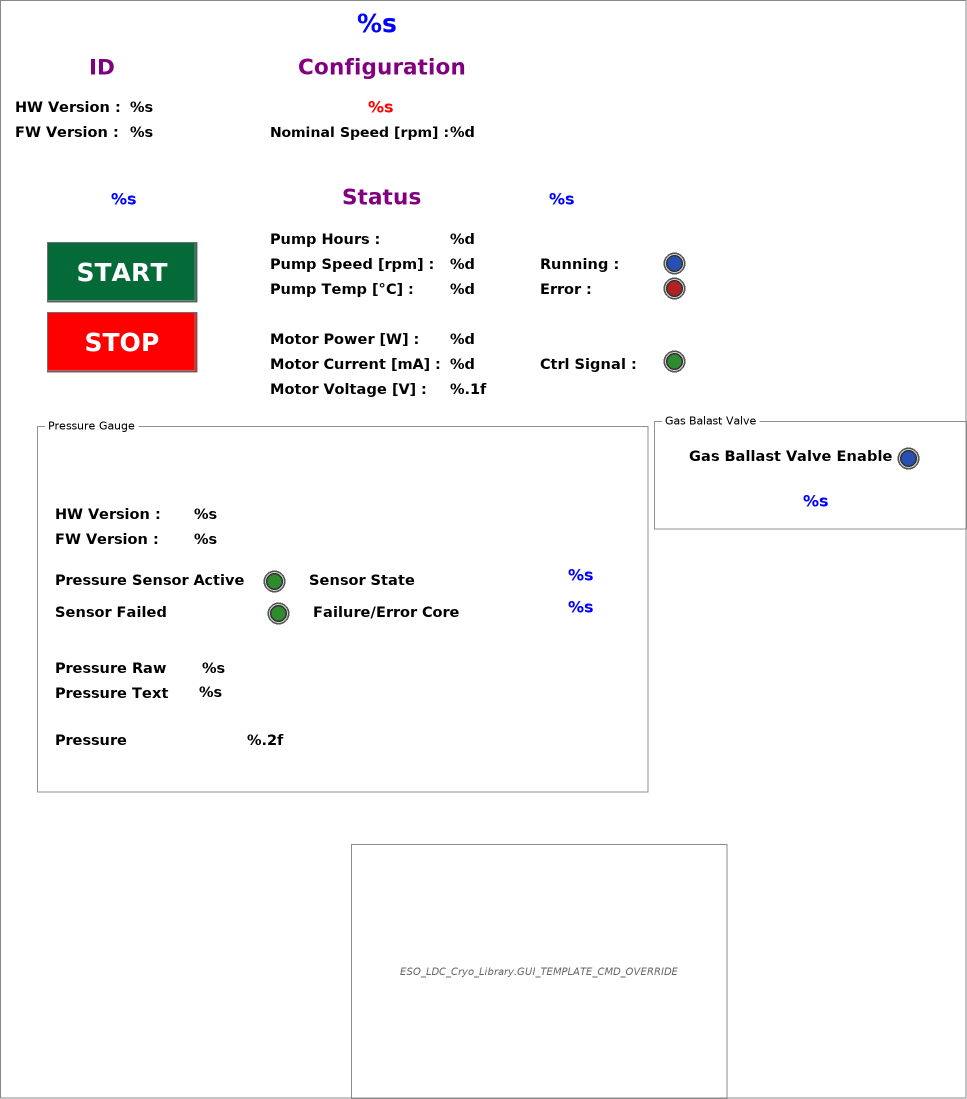
VISUALIZATION TEMPLATE_NOTT_PUMPS  // 967x1099
VAR_IN_OUT
	m_Instance:	FB_NOTT_PUMP_HICUBE_80_NEO;
	m_bEnable:	BOOL;	// Flag to start/stop the pump
	
END_VAR
    Rectangle (27,52 150x30), "ID"
    Rectangle (292,52 180x30), "Configuration"
    Rectangle (307,182 150x30), "Status"
    Lamp1 (662,251 25x25), tooltip "pump speed > 0 rpm", variable: m_Instance.stat.bMoving, style: Lamp-Lamp1-Blue
    Lamp1 (662,276 25x25), tooltip "presence of a warning", variable: m_Instance.stat.bFailure, style: Lamp-Lamp1-Red
    Rectangle (537,249 110x30), "Running :"
    Rectangle (537,274 110x30), "Error :"
    Rectangle (267,117 180x30), "Nominal Speed [rpm] :"
    Rectangle (267,224 180x30), "Pump Hours :"
    Rectangle (447,117 70x30), "%d", text variable: m_Instance.stat.nNominalSpeed
    Rectangle (447,224 70x30), "%d", text variable: m_Instance.stat.nPumpHours
    Rectangle (267,249 180x30), "Pump Speed [rpm] :"
    Rectangle (447,249 70x30), "%d", text variable: m_Instance.stat.nPumpSpeed
    Rectangle (267,274 180x30), "Pump Temp [°C] :"
    Rectangle (447,274 70x30), "%d", text variable: m_Instance.stat.nPumpTemp
    Rectangle (267,349 180x30), "Motor Current [mA] :"
    Rectangle (447,349 70x30), "%d", text variable: m_Instance.stat.nMotorCurr
    Rectangle (267,374 180x30), "Motor Voltage [V] :"
    Rectangle (447,374 70x30), "%.1f", text variable: m_Instance.stat.lrMotorVolt
    Rectangle (262,8 230x30), "%s", text variable: m_Instance.in_sName
    Rectangle (271,92 220x30), "%s", tooltip "Control Mode", text variable: m_Instance.stat.sCtrlViaInt
    Rectangle (127,92 130x30), "%s", tooltip "HW Version", text variable: m_Instance.stat.sHwVersion
    Rectangle (127,117 130x30), "%s", tooltip "FW Version", text variable: m_Instance.stat.sFwVersion
    Button (47,242 150x60), "START"
        OnMouseClick: execute { m_bEnable := TRUE; }
    Button (47,312 150x60), "STOP"
        OnMouseClick: execute { m_bEnable := FALSE; }
    Lamp1 (662,349 25x25), tooltip "If ON, control output signal is active.", variable: m_Instance.q_bStart, style: Lamp-Lamp1-Green
    Rectangle (537,349 110x30), "Ctrl Signal :"
    Rectangle (439,184 246x30), "%s", tooltip "Pump State", text variable: m_Instance.stat.sPumpState
    Rectangle (74,184 100x30), "%s", tooltip "Error Status", text variable: m_Instance.stat.sFailureCode
    Rectangle (267,324 180x30), "Motor Power [W] :"
    Rectangle (447,324 70x30), "%d", text variable: m_Instance.stat.nElecPower
    Rectangle (12,92 110x30), "HW Version :"
    Rectangle (12,117 110x30), "FW Version :"
    Frame (351,844 376x255)
        shows ESO_LDC_Cryo_Library.GUI_TEMPLATE_CMD_OVERRIDE(m_Cmd := MAIN.nott_cryo_ctrl.evac.ctrl.cor_PVP)
    GroupBox (37,418 611x374), "Pressure Gauge"
        Lamp1 (225,151 25x25), tooltip "Pressure Sensor ON", variable: m_Instance.stat.PresSens_bSensorOn, style: Lamp-Lamp1-Green
        Rectangle (15,147 254x30), "Pressure Sensor Active"
        Lamp1 (229,183 25x25), tooltip "Pressure Sensor ON", variable: m_Instance.stat.PresSens_bFailure, style: Lamp-Lamp1-Green
        Rectangle (269,147 254x30), "Sensor State"
        Rectangle (450,174 188x30), "%s", tooltip "Error Status", text variable: m_Instance.stat.PresSens_sFailureCode
        Rectangle (273,179 254x30), "Failure/Error Core"
        Rectangle (15,179 254x30), "Sensor Failed"
        Rectangle (450,142 188x30), "%s", tooltip "Error Status", text variable: m_Instance.stat.PresSens_sSensorState
        Rectangle (15,81 110x30), "HW Version :"
        Rectangle (154,81 130x30), "%s", tooltip "HW Version", text variable: m_Instance.stat.PresSens_sHwVersion
        Rectangle (154,106 130x30), "%s", tooltip "FW Version", text variable: m_Instance.stat.PresSens_sFwVersion
        Rectangle (15,106 110x30), "FW Version :"
        Rectangle (15,235 138x30), "Pressure Raw"
        Rectangle (162,235 130x30), "%s", tooltip "HW Version", text variable: m_Instance.stat.PresSens_sPressureRaw
        Rectangle (159,259 130x30), "%s", tooltip "FW Version", text variable: m_Instance.stat.PresSens_sPressureText
        Rectangle (15,260 142x30), "Pressure Text"
        Rectangle (15,307 180x30), "Pressure"
        Rectangle (207,307 197x30), "%.2f", text variable: m_Instance.stat.PresSens_lrPressure_hPa
    GroupBox (654,413 313x116), "Gas Balast Valve"
        Rectangle (39,73 246x30), "%s", tooltip "Gas Ballast valve status", text variable: m_Instance.stat.sGasBallastMode
        Lamp1 (242,33 25x25), tooltip "If ON, control output signal is active.", variable: m_Instance.stat.bGasBallastEnabled, style: Lamp-Lamp1-Blue
        Rectangle (32,28 211x30), "Gas Ballast Valve Enable"
END_VISUALIZATION

(* stored: Version 1.1.0.1, ProductVersion 3.1.4026.18
   Visu TEMPLATE_NOTT_PUMPS: Id {867471d6-c275-499d-b34c-834feb996f36} *)
